Yaskawa INFORM job: engine_cylinder_program.JBI

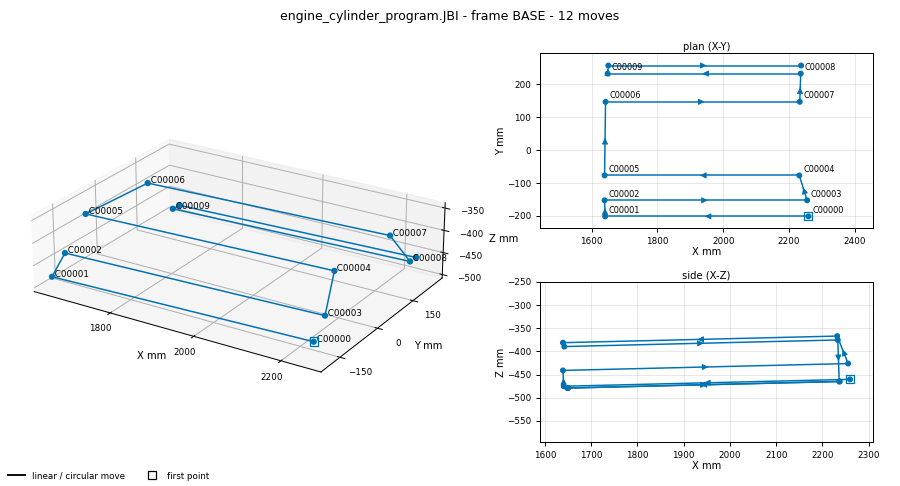
[picture p0: tool path of engine_cylinder_program.JBI in frame BASE, 12 of 15 moves have a stored position in this frame; points joined in program order, loops and branches not executed]
/JOB
//NAME engine_cylinder_program
//POS
///NPOS 12,0,12,0,0,0
///TOOL 0
///POSTYPE BASE
///RECTAN
///RCONF 0,0,0,0,0,0,0,0,0,0,0,0,0,0,0,0,0,0,0,0,0,0,0,0
C00000=2259.558718,-201.473124,-460.462407,175.000000,-60.000000,89.501928
C00001=1640.650651,-201.473123,-475.354673,175.000000,-60.000000,89.501928
C00002=1639.034045,-152.587115,-441.165198,175.000000,-50.331107,88.856602
C00003=2255.477092,-152.587115,-426.332245,175.000000,-50.331107,88.856602
C00004=2231.845655,-76.962491,-366.923754,-153.486424,-5.000000,-5.000000
C00005=1639.048457,-76.962491,-381.187737,-153.486424,-5.000000,-5.000000
C00006=1641.999546,147.195114,-389.560984,175.000000,-30.842932,-87.690586
C00007=2233.134188,147.195113,-375.337006,175.000000,-30.842932,-87.690586
C00008=2236.157256,233.185375,-465.043119,-175.000000,-61.646803,-89.255995
C00009=1648.365262,233.185375,-479.186666,-175.000000,-61.646803,-89.255995
C00010=1650.455017,257.644472,-479.289597,175.000000,-60.000000,-89.582026
C00011=2237.322706,257.644472,-465.168291,175.000000,-60.000000,-89.582026
///POSTYPE PULSE
///PULSE
EX00000=178176.0
///POSTYPE PULSE
///PULSE
EC00000=178176.0
EC00001=178176.0
EC00002=178176.0
EC00003=178176.0
EC00004=178176.0
EC00005=178176.0
EC00006=178176.0
EC00007=178176.0
EC00008=178176.0
EC00009=178176.0
EC00010=178176.0
EC00011=178176.0
//INST
///DATE 2023/08/16 18:17
///ATTR SC,RW,RJ
////FRAME BASE
///GROUP1 RB1,ST1
NOP
MOVJ P009 EX000 VJ=15.00
MOVJ C00000 EC00000 VJ=15.0
CALL JOB:SPYON
MOVL C00001 EC00001 V=150.0
MOVL C00002 EC00002 V=150.0
MOVL C00003 EC00003 V=150.0
MOVL C00004 EC00004 V=150.0
MOVL C00005 EC00005 V=150.0
MOVL C00006 EC00006 V=150.0
MOVL C00007 EC00007 V=150.0
MOVL C00008 EC00008 V=150.0
MOVL C00009 EC00009 V=150.0
MOVL C00010 EC00010 V=150.0
MOVL C00011 EC00011 V=150.0
CALL JOB:SPYOF
MOVJ P009 VJ=15.00
MOVL P009 EX00000 V=150.0
END
